// TwinCAT 3 PLC project Untitled1
// ProgramVersion: 3.1.4024.0
// libraries:
//   Tc2_Standard, * (Beckhoff Automation GmbH)
//   Tc2_System, * (Beckhoff Automation GmbH)
//   Tc3_Module, * (Beckhoff Automation GmbH)
// project tree:
//   / PlcTask.TcTTO
//   POUs/ CD_Observer.TcCD (not stored), FB_Display.TcPOU, FB_Station.TcPOU, ITF_Observable.TcIO, ITF_Observer.TcIO, MAIN.TcPOU
// real-time tasks:
//   TASK PlcTask: cycle T#10ms, priority 20, ADS port 350

CONFIGURATION Untitled1
    RESOURCE PLC ON TwinCAT3
        TASK PlcTask(INTERVAL := T#10ms, PRIORITY := 20);
        PROGRAM MAIN WITH PlcTask : MAIN;
    END_RESOURCE
END_CONFIGURATION

// ---- POUs/ITF_Observable.TcIO
INTERFACE ITF_Observable

METHOD notifyObserver : BOOL
VAR_INPUT
END_VAR
END_METHOD

METHOD registerObserver : BOOL
VAR_INPUT
	Observer : ITF_Observer;
END_VAR
END_METHOD

METHOD removeObserver : BOOL
VAR_INPUT
	Observer : ITF_Observer;
END_VAR
END_METHOD

END_INTERFACE

// ---- POUs/ITF_Observer.TcIO
INTERFACE ITF_Observer

PROPERTY ID : udint
GET
END_GET
SET
END_SET
END_PROPERTY

METHOD update : BOOL
VAR_INPUT
	Station : REFERENCE TO FB_Station;
END_VAR
END_METHOD

END_INTERFACE

// ---- POUs/MAIN.TcPOU
PROGRAM MAIN
VAR
	Initialized : BOOL;
	Station		: FB_Station;
	Display1	: FB_Display;
	Display2	: FB_Display;
	data		: INT;
	add1		: BOOL;
	add2		: BOOL;
	remove1		: BOOL;
	remove2		: BOOL;
END_VAR

//add Observers to Observable on startup
IF NOT Initialized THEN
	Station.registerObserver(Display1);
	Station.registerObserver(Display2);
	Initialized := TRUE;
END_IF

//remove observer
IF remove1 THEN
	remove1 := FALSE;
	Station.removeObserver(Display1);
END_IF

IF remove2 THEN
	remove2 := FALSE;
	Station.removeObserver(Display2);
END_IF

//add observer
IF add1 THEN
	add1 := FALSE;
	Station.registerObserver(Display1);
END_IF

IF add2 THEN
	add2 := FALSE;
	Station.registerObserver(Display2);
END_IF

//update code in all FBs
Station.CyclicLogic();
Display1.CyclicLogic();
Display2.CyclicLogic();

//Change this value for testing
Station.Data := data;

END_PROGRAM

// ---- POUs/FB_Station.TcPOU
FUNCTION_BLOCK FB_Station IMPLEMENTS ITF_Observable
VAR
	//ITF_Observable
	_Observers : ARRAY[1..2] OF ITF_Observer;
	_data	   : INT;
	prevData   : int;
END_VAR

METHOD CyclicLogic : BOOL
VAR
	dataChanged : BOOL;
END_VAR
//Monitor for change in data
IF data <> prevData THEN
	dataChanged := TRUE;
	prevData	:= Data;
END_IF

IF dataChanged THEN
	notifyObserver();
END_IF
END_METHOD

PROPERTY Data : int
GET
Data := _data;
END_GET
SET
_data := Data;
END_SET
END_PROPERTY

METHOD notifyObserver : BOOL
VAR
	i : UDINT;
END_VAR
FOR i := 1 TO 2 DO
	IF _Observers[i] <> 0 THEN
		_Observers[i].update(THIS^); //Call the update method of the observer and pass a reference to the Observable
	END_IF
END_FOR
END_METHOD

METHOD registerObserver : BOOL
VAR_INPUT
	Observer : ITF_Observer;
END_VAR

VAR
	i : UDINT;
END_VAR
//Find the first available array location and store a reference to the Observer there
FOR i := 1 TO 2 DO
	IF _Observers[i] = 0 THEN
		_Observers[i] := Observer;
		Observer.ID	  := i; //Send the location within the array back to the Observer, so it can pass the ID back when removing itself
		EXIT;
	END_IF
END_FOR
END_METHOD

METHOD removeObserver : BOOL
VAR_INPUT
	Observer : ITF_Observer;
END_VAR
//Check for valid reference
IF Observer <> 0 AND _Observers[Observer.ID] <> 0 THEN
	_Observers[Observer.ID] := 0; //Clear the array position
	Observer.ID				:= 0; //send back a 0 so the Observer knows it is no longer Observing
END_IF
END_METHOD

END_FUNCTION_BLOCK

// ---- POUs/FB_Display.TcPOU
FUNCTION_BLOCK FB_Display IMPLEMENTS ITF_Observer
VAR
	data : INT; //updated from the Observable
	_ID	 : udint; //set by the Observable
END_VAR

METHOD CyclicLogic : BOOL
VAR_INPUT
END_VAR
END_METHOD

PROPERTY ID : udint
GET
ID := _ID;
END_GET
SET
_ID := ID;
END_SET
END_PROPERTY

METHOD update : BOOL
VAR_INPUT
	Station : REFERENCE TO FB_Station;
END_VAR
data := Station.Data; //Read what you want from the Observable4
END_METHOD

END_FUNCTION_BLOCK
